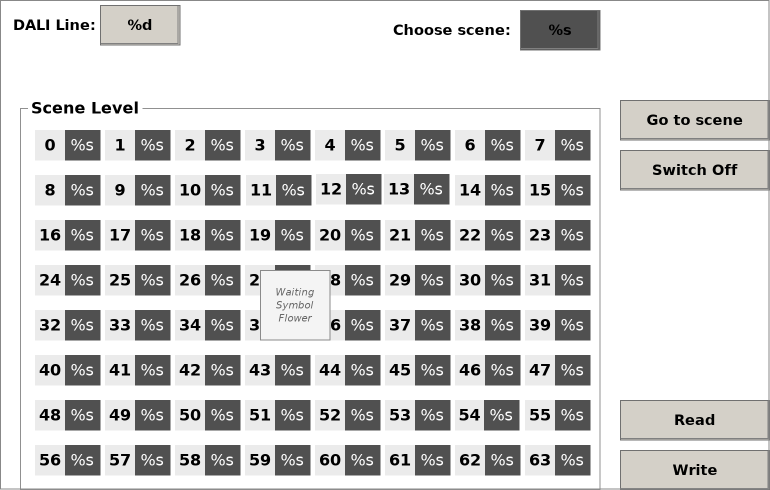
VISUALIZATION Visu_Part102Scenes  // 770x490
    GroupBox (20,100 580x390), "Scene Level"
        Group (85,30 65x30)
            Textfield (0,0 30x30), "1"
            Textfield (30,0 35x30), "%s", text variable: DALI_Commissioning.fbPart102Scenes.aScene[1], input disabled if: DALI_Commissioning.fbPart102Scenes.aNoShortAddress[1]
                p55702900: DALI_Commissioning.fbPart102Scenes.aFont[1]
                OnMouseClick: write the text variable via Default, min 0, max 255, title "Scene Value"
        Group (505,30 65x30)
            Textfield (0,0 30x30), "7"
            Textfield (30,0 35x30), "%s", text variable: DALI_Commissioning.fbPart102Scenes.aScene[7], input disabled if: DALI_Commissioning.fbPart102Scenes.aNoShortAddress[7]
                p55702900: DALI_Commissioning.fbPart102Scenes.aFont[7]
                OnMouseClick: write the text variable via Default, min 0, max 255, title "Scene Value"
        Group (435,30 65x30)
            Textfield (0,0 30x30), "6"
            Textfield (30,0 35x30), "%s", text variable: DALI_Commissioning.fbPart102Scenes.aScene[6], input disabled if: DALI_Commissioning.fbPart102Scenes.aNoShortAddress[6]
                p55702900: DALI_Commissioning.fbPart102Scenes.aFont[6]
                OnMouseClick: write the text variable via Default, min 0, max 255, title "Scene Value"
        Group (365,30 65x30)
            Textfield (0,0 30x30), "5"
            Textfield (30,0 35x30), "%s", text variable: DALI_Commissioning.fbPart102Scenes.aScene[5], input disabled if: DALI_Commissioning.fbPart102Scenes.aNoShortAddress[5]
                p55702900: DALI_Commissioning.fbPart102Scenes.aFont[5]
                OnMouseClick: write the text variable via Default, min 0, max 255, title "Scene Value"
        Group (295,30 65x30)
            Textfield (0,0 30x30), "4"
            Textfield (30,0 35x30), "%s", text variable: DALI_Commissioning.fbPart102Scenes.aScene[4], input disabled if: DALI_Commissioning.fbPart102Scenes.aNoShortAddress[4]
                p55702900: DALI_Commissioning.fbPart102Scenes.aFont[4]
                OnMouseClick: write the text variable via Default, min 0, max 255, title "Scene Value"
        Group (225,30 65x30)
            Textfield (0,0 30x30), "3"
            Textfield (30,0 35x30), "%s", text variable: DALI_Commissioning.fbPart102Scenes.aScene[3], input disabled if: DALI_Commissioning.fbPart102Scenes.aNoShortAddress[3]
                p55702900: DALI_Commissioning.fbPart102Scenes.aFont[3]
                OnMouseClick: write the text variable via Default, min 0, max 255, title "Scene Value"
        Group (155,30 65x30)
            Textfield (0,0 30x30), "2"
            Textfield (30,0 35x30), "%s", text variable: DALI_Commissioning.fbPart102Scenes.aScene[2], input disabled if: DALI_Commissioning.fbPart102Scenes.aNoShortAddress[2]
                p55702900: DALI_Commissioning.fbPart102Scenes.aFont[2]
                OnMouseClick: write the text variable via Default, min 0, max 255, title "Scene Value"
        Group (15,75 65x30)
            Textfield (0,0 30x30), "8"
            Textfield (30,0 35x30), "%s", text variable: DALI_Commissioning.fbPart102Scenes.aScene[8], input disabled if: DALI_Commissioning.fbPart102Scenes.aNoShortAddress[8]
                p55702900: DALI_Commissioning.fbPart102Scenes.aFont[8]
                OnMouseClick: write the text variable via Default, min 0, max 255, title "Scene Value"
        Group (15,120 65x30)
            Textfield (0,0 30x30), "16"
            Textfield (30,0 35x30), "%s", text variable: DALI_Commissioning.fbPart102Scenes.aScene[16], input disabled if: DALI_Commissioning.fbPart102Scenes.aNoShortAddress[16]
                p55702900: DALI_Commissioning.fbPart102Scenes.aFont[16]
                OnMouseClick: write the text variable via Default, min 0, max 255, title "Scene Value"
        Group (15,165 65x30)
            Textfield (0,0 30x30), "24"
            Textfield (30,0 35x30), "%s", text variable: DALI_Commissioning.fbPart102Scenes.aScene[24], input disabled if: DALI_Commissioning.fbPart102Scenes.aNoShortAddress[24]
                p55702900: DALI_Commissioning.fbPart102Scenes.aFont[24]
                OnMouseClick: write the text variable via Default, min 0, max 255, title "Scene Value"
        Group (15,210 65x30)
            Textfield (0,0 30x30), "32"
            Textfield (30,0 35x30), "%s", text variable: DALI_Commissioning.fbPart102Scenes.aScene[32], input disabled if: DALI_Commissioning.fbPart102Scenes.aNoShortAddress[32]
                p55702900: DALI_Commissioning.fbPart102Scenes.aFont[32]
                OnMouseClick: write the text variable via Default, min 0, max 255, title "Scene Value"
        Group (15,255 65x30)
            Textfield (0,0 30x30), "40"
            Textfield (30,0 35x30), "%s", text variable: DALI_Commissioning.fbPart102Scenes.aScene[40], input disabled if: DALI_Commissioning.fbPart102Scenes.aNoShortAddress[40]
                p55702900: DALI_Commissioning.fbPart102Scenes.aFont[40]
                OnMouseClick: write the text variable via Default, min 0, max 255, title "Scene Value"
        Group (15,300 65x30)
            Textfield (0,0 30x30), "48"
            Textfield (30,0 35x30), "%s", text variable: DALI_Commissioning.fbPart102Scenes.aScene[48], input disabled if: DALI_Commissioning.fbPart102Scenes.aNoShortAddress[48]
                p55702900: DALI_Commissioning.fbPart102Scenes.aFont[48]
                OnMouseClick: write the text variable via Default, min 0, max 255, title "Scene Value"
        Group (15,345 65x30)
            Textfield (0,0 30x30), "56"
            Textfield (30,0 35x30), "%s", text variable: DALI_Commissioning.fbPart102Scenes.aScene[56], input disabled if: DALI_Commissioning.fbPart102Scenes.aNoShortAddress[56]
                p55702900: DALI_Commissioning.fbPart102Scenes.aFont[56]
                OnMouseClick: write the text variable via Default, min 0, max 255, title "Scene Value"
        Group (85,75 65x30)
            Textfield (0,0 30x30), "9"
            Textfield (30,0 35x30), "%s", text variable: DALI_Commissioning.fbPart102Scenes.aScene[9], input disabled if: DALI_Commissioning.fbPart102Scenes.aNoShortAddress[9]
                p55702900: DALI_Commissioning.fbPart102Scenes.aFont[9]
                OnMouseClick: write the text variable via Default, min 0, max 255, title "Scene Value"
        Group (155,75 65x30)
            Textfield (0,0 30x30), "10"
            Textfield (30,0 35x30), "%s", text variable: DALI_Commissioning.fbPart102Scenes.aScene[10], input disabled if: DALI_Commissioning.fbPart102Scenes.aNoShortAddress[10]
                p55702900: DALI_Commissioning.fbPart102Scenes.aFont[10]
                OnMouseClick: write the text variable via Default, min 0, max 255, title "Scene Value"
        Group (226,75 65x30)
            Textfield (0,0 30x30), "11"
            Textfield (30,0 35x30), "%s", text variable: DALI_Commissioning.fbPart102Scenes.aScene[11], input disabled if: DALI_Commissioning.fbPart102Scenes.aNoShortAddress[11]
                p55702900: DALI_Commissioning.fbPart102Scenes.aFont[11]
                OnMouseClick: write the text variable via Default, min 0, max 255, title "Scene Value"
        Group (296,74 65x30)
            Textfield (0,0 30x30), "12"
            Textfield (30,0 35x30), "%s", text variable: DALI_Commissioning.fbPart102Scenes.aScene[12], input disabled if: DALI_Commissioning.fbPart102Scenes.aNoShortAddress[12]
                p55702900: DALI_Commissioning.fbPart102Scenes.aFont[12]
                OnMouseClick: write the text variable via Default, min 0, max 255, title "Scene Value"
        Group (364,74 65x30)
            Textfield (0,0 30x30), "13"
            Textfield (30,0 35x30), "%s", text variable: DALI_Commissioning.fbPart102Scenes.aScene[13], input disabled if: DALI_Commissioning.fbPart102Scenes.aNoShortAddress[13]
                p55702900: DALI_Commissioning.fbPart102Scenes.aFont[13]
                OnMouseClick: write the text variable via Default, min 0, max 255, title "Scene Value"
        Group (435,75 65x30)
            Textfield (0,0 30x30), "14"
            Textfield (30,0 35x30), "%s", text variable: DALI_Commissioning.fbPart102Scenes.aScene[14], input disabled if: DALI_Commissioning.fbPart102Scenes.aNoShortAddress[14]
                p55702900: DALI_Commissioning.fbPart102Scenes.aFont[14]
                OnMouseClick: write the text variable via Default, min 0, max 255, title "Scene Value"
        Group (505,75 65x30)
            Textfield (0,0 30x30), "15"
            Textfield (30,0 35x30), "%s", text variable: DALI_Commissioning.fbPart102Scenes.aScene[15], input disabled if: DALI_Commissioning.fbPart102Scenes.aNoShortAddress[15]
                p55702900: DALI_Commissioning.fbPart102Scenes.aFont[15]
                OnMouseClick: write the text variable via Default, min 0, max 255, title "Scene Value"
        Group (85,120 65x30)
            Textfield (0,0 30x30), "17"
            Textfield (30,0 35x30), "%s", text variable: DALI_Commissioning.fbPart102Scenes.aScene[17], input disabled if: DALI_Commissioning.fbPart102Scenes.aNoShortAddress[17]
                p55702900: DALI_Commissioning.fbPart102Scenes.aFont[17]
                OnMouseClick: write the text variable via Default, min 0, max 255, title "Scene Value"
        Group (155,120 65x30)
            Textfield (0,0 30x30), "18"
            Textfield (30,0 35x30), "%s", text variable: DALI_Commissioning.fbPart102Scenes.aScene[18], input disabled if: DALI_Commissioning.fbPart102Scenes.aNoShortAddress[18]
                p55702900: DALI_Commissioning.fbPart102Scenes.aFont[18]
                OnMouseClick: write the text variable via Default, min 0, max 255, title "Scene Value"
        Group (225,120 65x30)
            Textfield (0,0 30x30), "19"
            Textfield (30,0 35x30), "%s", text variable: DALI_Commissioning.fbPart102Scenes.aScene[19], input disabled if: DALI_Commissioning.fbPart102Scenes.aNoShortAddress[19]
                p55702900: DALI_Commissioning.fbPart102Scenes.aFont[19]
                OnMouseClick: write the text variable via Default, min 0, max 255, title "Scene Value"
        Group (295,120 65x30)
            Textfield (0,0 30x30), "20"
            Textfield (30,0 35x30), "%s", text variable: DALI_Commissioning.fbPart102Scenes.aScene[20], input disabled if: DALI_Commissioning.fbPart102Scenes.aNoShortAddress[20]
                p55702900: DALI_Commissioning.fbPart102Scenes.aFont[20]
                OnMouseClick: write the text variable via Default, min 0, max 255, title "Scene Value"
        Group (365,120 65x30)
            Textfield (0,0 30x30), "21"
            Textfield (30,0 35x30), "%s", text variable: DALI_Commissioning.fbPart102Scenes.aScene[21], input disabled if: DALI_Commissioning.fbPart102Scenes.aNoShortAddress[21]
                p55702900: DALI_Commissioning.fbPart102Scenes.aFont[21]
                OnMouseClick: write the text variable via Default, min 0, max 255, title "Scene Value"
        Group (435,120 65x30)
            Textfield (0,0 30x30), "22"
            Textfield (30,0 35x30), "%s", text variable: DALI_Commissioning.fbPart102Scenes.aScene[22], input disabled if: DALI_Commissioning.fbPart102Scenes.aNoShortAddress[22]
                p55702900: DALI_Commissioning.fbPart102Scenes.aFont[22]
                OnMouseClick: write the text variable via Default, min 0, max 255, title "Scene Value"
        Group (505,120 65x30)
            Textfield (0,0 30x30), "23"
            Textfield (30,0 35x30), "%s", text variable: DALI_Commissioning.fbPart102Scenes.aScene[23], input disabled if: DALI_Commissioning.fbPart102Scenes.aNoShortAddress[23]
                p55702900: DALI_Commissioning.fbPart102Scenes.aFont[23]
                OnMouseClick: write the text variable via Default, min 0, max 255, title "Scene Value"
        Group (85,165 65x30)
            Textfield (0,0 30x30), "25"
            Textfield (30,0 35x30), "%s", text variable: DALI_Commissioning.fbPart102Scenes.aScene[25], input disabled if: DALI_Commissioning.fbPart102Scenes.aNoShortAddress[25]
                p55702900: DALI_Commissioning.fbPart102Scenes.aFont[25]
                OnMouseClick: write the text variable via Default, min 0, max 255, title "Scene Value"
        Group (155,165 65x30)
            Textfield (0,0 30x30), "26"
            Textfield (30,0 35x30), "%s", text variable: DALI_Commissioning.fbPart102Scenes.aScene[26], input disabled if: DALI_Commissioning.fbPart102Scenes.aNoShortAddress[26]
                p55702900: DALI_Commissioning.fbPart102Scenes.aFont[26]
                OnMouseClick: write the text variable via Default, min 0, max 255, title "Scene Value"
        Group (225,165 65x30)
            Textfield (0,0 30x30), "27"
            Textfield (30,0 35x30), "%s", text variable: DALI_Commissioning.fbPart102Scenes.aScene[27], input disabled if: DALI_Commissioning.fbPart102Scenes.aNoShortAddress[27]
                p55702900: DALI_Commissioning.fbPart102Scenes.aFont[27]
                OnMouseClick: write the text variable via Default, min 0, max 255, title "Scene Value"
        Group (295,165 65x30)
            Textfield (0,0 30x30), "28"
            Textfield (30,0 35x30), "%s", text variable: DALI_Commissioning.fbPart102Scenes.aScene[28], input disabled if: DALI_Commissioning.fbPart102Scenes.aNoShortAddress[28]
                p55702900: DALI_Commissioning.fbPart102Scenes.aFont[28]
                OnMouseClick: write the text variable via Default, min 0, max 255, title "Scene Value"
        Group (365,165 65x30)
            Textfield (0,0 30x30), "29"
            Textfield (30,0 35x30), "%s", text variable: DALI_Commissioning.fbPart102Scenes.aScene[29], input disabled if: DALI_Commissioning.fbPart102Scenes.aNoShortAddress[29]
                p55702900: DALI_Commissioning.fbPart102Scenes.aFont[29]
                OnMouseClick: write the text variable via Default, min 0, max 255, title "Scene Value"
        Group (435,165 65x30)
            Textfield (0,0 30x30), "30"
            Textfield (30,0 35x30), "%s", text variable: DALI_Commissioning.fbPart102Scenes.aScene[30], input disabled if: DALI_Commissioning.fbPart102Scenes.aNoShortAddress[30]
                p55702900: DALI_Commissioning.fbPart102Scenes.aFont[30]
                OnMouseClick: write the text variable via Default, min 0, max 255, title "Scene Value"
        Group (505,165 65x30)
            Textfield (0,0 30x30), "31"
            Textfield (30,0 35x30), "%s", text variable: DALI_Commissioning.fbPart102Scenes.aScene[31], input disabled if: DALI_Commissioning.fbPart102Scenes.aNoShortAddress[31]
                p55702900: DALI_Commissioning.fbPart102Scenes.aFont[31]
                OnMouseClick: write the text variable via Default, min 0, max 255, title "Scene Value"
        Group (85,210 65x30)
            Textfield (0,0 30x30), "33"
            Textfield (30,0 35x30), "%s", text variable: DALI_Commissioning.fbPart102Scenes.aScene[33], input disabled if: DALI_Commissioning.fbPart102Scenes.aNoShortAddress[32]
                p55702900: DALI_Commissioning.fbPart102Scenes.aFont[33]
                OnMouseClick: write the text variable via Default, min 0, max 255, title "Scene Value"
        Group (155,210 65x30)
            Textfield (0,0 30x30), "34"
            Textfield (30,0 35x30), "%s", text variable: DALI_Commissioning.fbPart102Scenes.aScene[34], input disabled if: DALI_Commissioning.fbPart102Scenes.aNoShortAddress[34]
                p55702900: DALI_Commissioning.fbPart102Scenes.aFont[34]
                OnMouseClick: write the text variable via Default, min 0, max 255, title "Scene Value"
        Group (295,210 65x30)
            Textfield (0,0 30x30), "36"
            Textfield (30,0 35x30), "%s", text variable: DALI_Commissioning.fbPart102Scenes.aScene[36], input disabled if: DALI_Commissioning.fbPart102Scenes.aNoShortAddress[36]
                p55702900: DALI_Commissioning.fbPart102Scenes.aFont[36]
                OnMouseClick: write the text variable via Default, min 0, max 255
        Group (365,210 65x30)
            Textfield (0,0 30x30), "37"
            Textfield (30,0 35x30), "%s", text variable: DALI_Commissioning.fbPart102Scenes.aScene[37], input disabled if: DALI_Commissioning.fbPart102Scenes.aNoShortAddress[37]
                p55702900: DALI_Commissioning.fbPart102Scenes.aFont[37]
                OnMouseClick: write the text variable via Default, min 0, max 255, title "Scene Value"
        Group (435,210 65x30)
            Textfield (0,0 30x30), "38"
            Textfield (30,0 35x30), "%s", text variable: DALI_Commissioning.fbPart102Scenes.aScene[38], input disabled if: DALI_Commissioning.fbPart102Scenes.aNoShortAddress[38]
                p55702900: DALI_Commissioning.fbPart102Scenes.aFont[38]
                OnMouseClick: write the text variable via Default, min 0, max 255, title "Scene Value"
        Group (505,210 65x30)
            Textfield (0,0 30x30), "39"
            Textfield (30,0 35x30), "%s", text variable: DALI_Commissioning.fbPart102Scenes.aScene[39], input disabled if: DALI_Commissioning.fbPart102Scenes.aNoShortAddress[39]
                p55702900: DALI_Commissioning.fbPart102Scenes.aFont[39]
                OnMouseClick: write the text variable via Default, min 0, max 255, title "Scene Value"
        Group (85,255 65x30)
            Textfield (0,0 30x30), "41"
            Textfield (30,0 35x30), "%s", text variable: DALI_Commissioning.fbPart102Scenes.aScene[41], input disabled if: DALI_Commissioning.fbPart102Scenes.aNoShortAddress[41]
                p55702900: DALI_Commissioning.fbPart102Scenes.aFont[41]
                OnMouseClick: write the text variable via Default, min 0, max 255, title "Scene Value"
        Group (155,255 65x30)
            Textfield (0,0 30x30), "42"
            Textfield (30,0 35x30), "%s", text variable: DALI_Commissioning.fbPart102Scenes.aScene[42], input disabled if: DALI_Commissioning.fbPart102Scenes.aNoShortAddress[42]
                p55702900: DALI_Commissioning.fbPart102Scenes.aFont[42]
                OnMouseClick: write the text variable via Default, min 0, max 255, title "Scene Value"
        Group (225,210 65x30)
            Textfield (0,0 30x30), "35"
            Textfield (30,0 35x30), "%s", text variable: DALI_Commissioning.fbPart102Scenes.aScene[35], input disabled if: DALI_Commissioning.fbPart102Scenes.aNoShortAddress[35]
                p55702900: DALI_Commissioning.fbPart102Scenes.aFont[35]
                OnMouseClick: write the text variable via Default, min 0, max 255, title "Scene Value"
        Group (225,255 65x30)
            Textfield (0,0 30x30), "43"
            Textfield (30,0 35x30), "%s", text variable: DALI_Commissioning.fbPart102Scenes.aScene[43], input disabled if: DALI_Commissioning.fbPart102Scenes.aNoShortAddress[43]
                p55702900: DALI_Commissioning.fbPart102Scenes.aFont[43]
                OnMouseClick: write the text variable via Default, min 0, max 255, title "Scene Value"
        Group (295,255 65x30)
            Textfield (0,0 30x30), "44"
            Textfield (30,0 35x30), "%s", text variable: DALI_Commissioning.fbPart102Scenes.aScene[44], input disabled if: DALI_Commissioning.fbPart102Scenes.aNoShortAddress[44]
                p55702900: DALI_Commissioning.fbPart102Scenes.aFont[44]
                OnMouseClick: write the text variable via Default, min 0, max 255, title "Scene Value"
        Group (365,255 65x30)
            Textfield (0,0 30x30), "45"
            Textfield (30,0 35x30), "%s", text variable: DALI_Commissioning.fbPart102Scenes.aScene[45], input disabled if: DALI_Commissioning.fbPart102Scenes.aNoShortAddress[45]
                p55702900: DALI_Commissioning.fbPart102Scenes.aFont[45]
                OnMouseClick: write the text variable via Default, min 0, max 255, title "Scene Value"
        Group (435,255 65x30)
            Textfield (0,0 30x30), "46"
            Textfield (30,0 35x30), "%s", text variable: DALI_Commissioning.fbPart102Scenes.aScene[46], input disabled if: DALI_Commissioning.fbPart102Scenes.aNoShortAddress[46]
                p55702900: DALI_Commissioning.fbPart102Scenes.aFont[46]
                OnMouseClick: write the text variable via Default, min 0, max 255, title "Scene Value"
        Group (505,255 65x30)
            Textfield (0,0 30x30), "47"
            Textfield (30,0 35x30), "%s", text variable: DALI_Commissioning.fbPart102Scenes.aScene[47], input disabled if: DALI_Commissioning.fbPart102Scenes.aNoShortAddress[47]
                p55702900: DALI_Commissioning.fbPart102Scenes.aFont[47]
                OnMouseClick: write the text variable via Default, min 0, max 255, title "Scene Value"
        Group (85,300 65x30)
            Textfield (0,0 30x30), "49"
            Textfield (30,0 35x30), "%s", text variable: DALI_Commissioning.fbPart102Scenes.aScene[49], input disabled if: DALI_Commissioning.fbPart102Scenes.aNoShortAddress[49]
                p55702900: DALI_Commissioning.fbPart102Scenes.aFont[49]
                OnMouseClick: write the text variable via Default, min 0, max 255, title "Scene Value"
        Group (155,300 65x30)
            Textfield (0,0 30x30), "50"
            Textfield (30,0 35x30), "%s", text variable: DALI_Commissioning.fbPart102Scenes.aScene[50], input disabled if: DALI_Commissioning.fbPart102Scenes.aNoShortAddress[50]
                p55702900: DALI_Commissioning.fbPart102Scenes.aFont[50]
                OnMouseClick: write the text variable via Default, min 0, max 255, title "Scene Value"
        Group (225,300 65x30)
            Textfield (0,0 30x30), "51"
            Textfield (30,0 35x30), "%s", text variable: DALI_Commissioning.fbPart102Scenes.aScene[51], input disabled if: DALI_Commissioning.fbPart102Scenes.aNoShortAddress[51]
                p55702900: DALI_Commissioning.fbPart102Scenes.aFont[51]
                OnMouseClick: write the text variable via Default, min 0, max 255, title "Scene Value"
        Group (295,300 65x30)
            Textfield (0,0 30x30), "52"
            Textfield (30,0 35x30), "%s", text variable: DALI_Commissioning.fbPart102Scenes.aScene[52], input disabled if: DALI_Commissioning.fbPart102Scenes.aNoShortAddress[52]
                p55702900: DALI_Commissioning.fbPart102Scenes.aFont[52]
                OnMouseClick: write the text variable via Default, min 0, max 255, title "Scene Value"
        Group (365,300 65x30)
            Textfield (0,0 30x30), "53"
            Textfield (30,0 35x30), "%s", text variable: DALI_Commissioning.fbPart102Scenes.aScene[53], input disabled if: DALI_Commissioning.fbPart102Scenes.aNoShortAddress[53]
                p55702900: DALI_Commissioning.fbPart102Scenes.aFont[53]
                OnMouseClick: write the text variable via Default, min 0, max 255, title "Scene Value"
        Group (435,300 64x30)
            Textfield (0,0 29x30), "54"
            Textfield (29,0 35x30), "%s", text variable: DALI_Commissioning.fbPart102Scenes.aScene[54], input disabled if: DALI_Commissioning.fbPart102Scenes.aNoShortAddress[54]
                p55702900: DALI_Commissioning.fbPart102Scenes.aFont[54]
                OnMouseClick: write the text variable via Default, min 0, max 255, title "Scene Value"
        Group (505,300 65x30)
            Textfield (0,0 30x30), "55"
            Textfield (30,0 35x30), "%s", text variable: DALI_Commissioning.fbPart102Scenes.aScene[55], input disabled if: DALI_Commissioning.fbPart102Scenes.aNoShortAddress[55]
                p55702900: DALI_Commissioning.fbPart102Scenes.aFont[55]
                OnMouseClick: write the text variable via Default, min 0, max 255, title "Scene Value"
        Group (85,345 65x30)
            Textfield (0,0 30x30), "57"
            Textfield (30,0 35x30), "%s", text variable: DALI_Commissioning.fbPart102Scenes.aScene[57], input disabled if: DALI_Commissioning.fbPart102Scenes.aNoShortAddress[57]
                p55702900: DALI_Commissioning.fbPart102Scenes.aFont[57]
                OnMouseClick: write the text variable via Default, min 0, max 255, title "Scene Value"
        Group (155,345 65x30)
            Textfield (0,0 30x30), "58"
            Textfield (30,0 35x30), "%s", text variable: DALI_Commissioning.fbPart102Scenes.aScene[58], input disabled if: DALI_Commissioning.fbPart102Scenes.aNoShortAddress[58]
                p55702900: DALI_Commissioning.fbPart102Scenes.aFont[58]
                OnMouseClick: write the text variable via Default, min 0, max 255, title "Scene Value"
        Group (225,345 65x30)
            Textfield (0,0 30x30), "59"
            Textfield (30,0 35x30), "%s", text variable: DALI_Commissioning.fbPart102Scenes.aScene[59], input disabled if: DALI_Commissioning.fbPart102Scenes.aNoShortAddress[59]
                p55702900: DALI_Commissioning.fbPart102Scenes.aFont[59]
                OnMouseClick: write the text variable via Default, min 0, max 255, title "Scene Value"
        Group (295,345 65x30)
            Textfield (0,0 30x30), "60"
            Textfield (30,0 35x30), "%s", text variable: DALI_Commissioning.fbPart102Scenes.aScene[60], input disabled if: DALI_Commissioning.fbPart102Scenes.aNoShortAddress[60]
                p55702900: DALI_Commissioning.fbPart102Scenes.aFont[60]
                OnMouseClick: write the text variable via Default, min 0, max 255, title "Scene Value"
        Group (365,345 65x30)
            Textfield (0,0 30x30), "61"
            Textfield (30,0 35x30), "%s", text variable: DALI_Commissioning.fbPart102Scenes.aScene[61], input disabled if: DALI_Commissioning.fbPart102Scenes.aNoShortAddress[61]
                p55702900: DALI_Commissioning.fbPart102Scenes.aFont[61]
                OnMouseClick: write the text variable via Default, min 0, max 255, title "Scene Value"
        Group (435,345 65x30)
            Textfield (0,0 30x30), "62"
            Textfield (30,0 35x30), "%s", text variable: DALI_Commissioning.fbPart102Scenes.aScene[62], input disabled if: DALI_Commissioning.fbPart102Scenes.aNoShortAddress[62]
                p55702900: DALI_Commissioning.fbPart102Scenes.aFont[62]
                OnMouseClick: write the text variable via Default, min 0, max 255, title "Scene Value"
        Group (505,345 65x30)
            Textfield (0,0 30x30), "63"
            Textfield (30,0 35x30), "%s", text variable: DALI_Commissioning.fbPart102Scenes.aScene[63], input disabled if: DALI_Commissioning.fbPart102Scenes.aNoShortAddress[63]
                p55702900: DALI_Commissioning.fbPart102Scenes.aFont[63]
                OnMouseClick: write the text variable via Default, min 0, max 255, title "Scene Value"
        WaitingSymbolFlower (240,170 70x70), invisible if: DALI_Commissioning.fbPart102Scenes.bHideWaitSymbol
        Group (15,30 65x30)
            Textfield (0,0 30x30), "0"
            Textfield (30,0 35x30), "%s", text variable: DALI_Commissioning.fbPart102Scenes.aScene[0], input disabled if: DALI_Commissioning.fbPart102Scenes.aNoShortAddress[0]
                p55702900: DALI_Commissioning.fbPart102Scenes.aFont[0]
                OnMouseClick: write the text variable via Default, min 0, max 255, title "Scene Value"
    Button (620,400 150x40), "Read"
        OnMouseClick: execute { DALI_Commissioning.fbPart102Scenes.bRead := TRUE; }
    Button (620,450 150x40), "Write"
        OnMouseClick: execute { DALI_Commissioning.fbPart102Scenes.bWrite := TRUE; }
    Button (620,100 150x40), "Go to scene"
        OnMouseClick: execute { DALI_Commissioning.fbPart102Scenes.bGoToScene := TRUE; }
    Button (620,150 150x40), "Switch Off"
        OnMouseClick: execute { DALI_Commissioning.fbPart102Scenes.bSwitchOff := TRUE; }
    Textfield (390,10 120x40), "Choose scene:"
    Button (520,10 80x40), "%s", text variable: DALI_Commissioning.fbPart102Scenes.nScene
        OnMouseClick: write the text variable via Default, min 0, max 15, title "Choose scene"
    Group (10,5 170x40)
        Textfield (0,0 110x40), "DALI Line:"
        Button (90,0 80x40), "%d", text variable: GVL_Internal.nDALILine
            OnMouseClick: write the text variable via Default, min 1, max 10, title "Choose line"
END_VISUALIZATION

(* stored: Version 1.1.0.1, ProductVersion 3.1.4024.12
   Visu Visu_Part102Scenes: Id {32879f24-5327-488d-a69f-4977bee7d53e} *)
